TYPE "udt_BimanualSts"
VERSION : 0.1
// Block: udt_BimanualSts
   STRUCT
      SafeMotion : Bool;
      Enable : Bool;
   END_STRUCT;

END_TYPE
